KUKA KRL program: chequeo_paleta.src, chequeo_paleta.dat

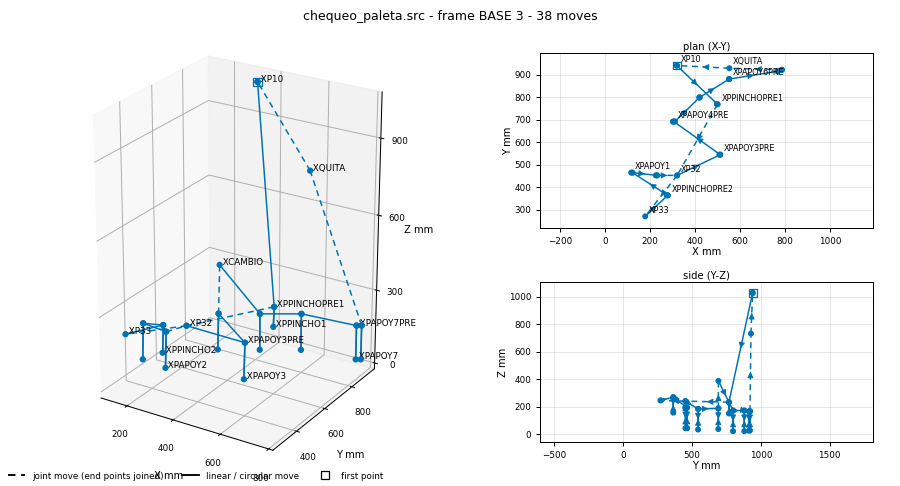
[picture p0: tool path of chequeo_paleta.src in frame BASE 3, 38 of 42 moves have a stored position in this frame; points joined in program order, loops and branches not executed]
--- chequeo_paleta.src ---
&ACCESS RVP
&REL 223
&COMMENT COGER ST121 RACK AZUL
&PARAM EDITMASK = *
&PARAM TEMPLATE = C:\KRC\Roboter\Template\vorgabe
&PARAM DISKPATH = KRC:\R1\Program\MAFELEC
DEF chequeo_paleta( )
;FOLD INI;%{PE}
  ;FOLD BASISTECH INI
    GLOBAL INTERRUPT DECL 3 WHEN $STOPMESS==TRUE DO IR_STOPM ( )
    INTERRUPT ON 3
    BAS (#INITMOV,0 )
  ;ENDFOLD (BASISTECH INI)
;FOLD SPOTTECH INI
USERSPOT(#INIT)
;ENDFOLD (SPOTTECH INI)
;FOLD GRIPPERTECH INI
USER_GRP(0,DUMMY,DUMMY,GDEFAULT)
;ENDFOLD (GRIPPERTECH INI)
;FOLD USER INI
INTERRUPT DECL 26 WHEN I_121R1S102 OR I_121R1S202 DO PARO_RAPIDO ()
INTERRUPT DECL 27 WHEN I_121R1S302 OR I_121R1S402 DO PARO_RAPIDO ()

    ;Make your modifications here

  ;ENDFOLD (USER INI)
;ENDFOLD (INI)
;################################################
; PROYECTO: PLANTA DE BATERIAS
; ROBOT: 121_R1 TERMINATOR
; PROGRAMA: Chequeo_paletas EN ST121
; PALETA MASTER NUMERO 20
; CREADO POR: Borja Carrion
; FECHA: 13-JULIO-2024
;################################################

Empujador(1,"R",FALSE)
Empujador(2,"R",FALSE)

;FOLD PTP HOME Vel=100 % DEFAULT;%{PE}%R 8.3.48,%MKUKATPBASIS,%CMOVE,%VPTP,%P 1:PTP, 2:HOME, 3:, 5:100, 7:DEFAULT
$BWDSTART=FALSE
PDAT_ACT=PDEFAULT
FDAT_ACT=FHOME
BAS(#PTP_PARAMS,100)
$H_POS=XHOME
PTP XHOME
;ENDFOLD
; FOLD ESPERA CONFIRMACION ENTRADA INSPECCION
WAIT FOR I_ST121_INSPECCION
; ENDFOLD

;FOLD PTP POS_ESPERA_ST121 Vel=100 % H Tool[9]:T_Gripper1_Vacio Base[0];%{PE}%R 8.3.48,%MKUKATPBASIS,%CMOVE,%VPTP,%P 1:PTP, 2:POS_ESPERA_ST121, 3:, 5:100, 7:H
$BWDSTART=FALSE
PDAT_ACT=PH
FDAT_ACT=FPOS_ESPERA_ST121
BAS(#PTP_PARAMS,100)
PTP XPOS_ESPERA_ST121
;ENDFOLD

; FOLD ESPERA CONFIRMACION ENTRADA INSPECCION
WAIT FOR I_ST121_INSPECCION
; ENDFOLD

; FOLD CONTROL DE ELEMENTOS MECANICOS EN REPOSO
;CONTROL DE AUSENCIA DE PIEZA EN GRIPPER
IF I_121R1S1000 THEN
HALT
ENDIF

;CONTROL APERTURA GRIPPER

IF (I_121R1S131B==FALSE) OR (I_121R1S132B==FALSE) OR (I_121R1S133B==FALSE) OR (I_121R1S134B==FALSE) THEN
Pines("R")
ENDIF

Empujador(1,"R",TRUE)
Empujador(2,"R",TRUE)
; ENDFOLD

;FOLD PTP P10 CONT Vel=100 % M Tool[9]:T_Gripper1_Vacio Base[3]:ST121;%{PE}%R 8.3.48,%MKUKATPBASIS,%CMOVE,%VPTP,%P 1:PTP, 2:P10, 3:C_DIS, 5:100, 7:M
$BWDSTART=FALSE
PDAT_ACT=PM
FDAT_ACT=FP10
BAS(#PTP_PARAMS,100)
PTP XP10 C_DIS
;ENDFOLD


; ANTES DE EMPEZAR EL CHEQUEO COLOCAR EL UTIL EN LA CLAMPA 3 (QUITAR TONILLO AZUL)
; ABRIR PUERTA DESCARGA MANUAL

; POSICIONES CHEQUEO PINCHOS

; PINCHO 1
;FOLD LIN PPINCHOPRE1 CONT Vel=0.09 m/s M Tool[9]:T_Gripper1_Vacio Base[3]:ST121;%{PE}%R 8.3.48,%MKUKATPBASIS,%CMOVE,%VLIN,%P 1:LIN, 2:PPINCHOPRE1, 3:C_DIS C_DIS, 5:0.09, 7:M
$BWDSTART=FALSE
LDAT_ACT=LM
FDAT_ACT=FPPINCHOPRE1
BAS(#CP_PARAMS,0.09)
LIN XPPINCHOPRE1 C_DIS C_DIS
;ENDFOLD
;FOLD LIN PPINCHO1 CONT Vel=0.02 m/s M Tool[9]:T_Gripper1_Vacio Base[3]:ST121;%{PE}%R 8.3.48,%MKUKATPBASIS,%CMOVE,%VLIN,%P 1:LIN, 2:PPINCHO1, 3:C_DIS C_DIS, 5:0.02, 7:M
$BWDSTART=FALSE
LDAT_ACT=LM
FDAT_ACT=FPPINCHO1
BAS(#CP_PARAMS,0.02)
LIN XPPINCHO1 C_DIS C_DIS
;ENDFOLD
;FOLD WAIT Time=0.5 sec;%{PE}%R 8.3.48,%MKUKATPBASIS,%CWAIT,%VWAIT,%P 3:0.5
WAIT SEC 0.5
;ENDFOLD
;FOLD LIN PPINCHOPRE1 CONT Vel=0.09 m/s M Tool[9]:T_Gripper1_Vacio Base[3]:ST121;%{PE}%R 8.3.48,%MKUKATPBASIS,%CMOVE,%VLIN,%P 1:LIN, 2:PPINCHOPRE1, 3:C_DIS C_DIS, 5:0.09, 7:M
$BWDSTART=FALSE
LDAT_ACT=LM
FDAT_ACT=FPPINCHOPRE1
BAS(#CP_PARAMS,0.09)
LIN XPPINCHOPRE1 C_DIS C_DIS
;ENDFOLD

; PINCHO 2
;FOLD PTP P32 CONT Vel=50 % M Tool[9]:T_Gripper1_Vacio Base[3]:ST121;%{PE}%R 8.3.48,%MKUKATPBASIS,%CMOVE,%VPTP,%P 1:PTP, 2:P32, 3:C_DIS, 5:50, 7:M
$BWDSTART=FALSE
PDAT_ACT=PM
FDAT_ACT=FP32
BAS(#PTP_PARAMS,50)
PTP XP32 C_DIS
;ENDFOLD
;FOLD PTP P33 CONT Vel=50 % M Tool[9]:T_Gripper1_Vacio Base[3]:ST121;%{PE}%R 8.3.48,%MKUKATPBASIS,%CMOVE,%VPTP,%P 1:PTP, 2:P33, 3:C_DIS, 5:50, 7:M
$BWDSTART=FALSE
PDAT_ACT=PM
FDAT_ACT=FP33
BAS(#PTP_PARAMS,50)
PTP XP33 C_DIS
;ENDFOLD
;FOLD LIN PPINCHOPRE2 CONT Vel=0.09 m/s M Tool[9]:T_Gripper1_Vacio Base[3]:ST121;%{PE}%R 8.3.48,%MKUKATPBASIS,%CMOVE,%VLIN,%P 1:LIN, 2:PPINCHOPRE2, 3:C_DIS C_DIS, 5:0.09, 7:M
$BWDSTART=FALSE
LDAT_ACT=LM
FDAT_ACT=FPPINCHOPRE2
BAS(#CP_PARAMS,0.09)
LIN XPPINCHOPRE2 C_DIS C_DIS
;ENDFOLD
;FOLD LIN PPINCHO2 CONT Vel=0.02 m/s M Tool[9]:T_Gripper1_Vacio Base[3]:ST121;%{PE}%R 8.3.48,%MKUKATPBASIS,%CMOVE,%VLIN,%P 1:LIN, 2:PPINCHO2, 3:C_DIS C_DIS, 5:0.02, 7:M
$BWDSTART=FALSE
LDAT_ACT=LM
FDAT_ACT=FPPINCHO2
BAS(#CP_PARAMS,0.02)
LIN XPPINCHO2 C_DIS C_DIS
;ENDFOLD
;FOLD WAIT Time=0.5 sec;%{PE}%R 8.3.48,%MKUKATPBASIS,%CWAIT,%VWAIT,%P 3:0.5
WAIT SEC 0.5
;ENDFOLD
;FOLD LIN PPINCHOPRE2 CONT Vel=0.09 m/s M Tool[9]:T_Gripper1_Vacio Base[3]:ST121;%{PE}%R 8.3.48,%MKUKATPBASIS,%CMOVE,%VLIN,%P 1:LIN, 2:PPINCHOPRE2, 3:C_DIS C_DIS, 5:0.09, 7:M
$BWDSTART=FALSE
LDAT_ACT=LM
FDAT_ACT=FPPINCHOPRE2
BAS(#CP_PARAMS,0.09)
LIN XPPINCHOPRE2 C_DIS C_DIS
;ENDFOLD

;FOLD WAIT Time=1 sec;%{PE}%R 8.3.48,%MKUKATPBASIS,%CWAIT,%VWAIT,%P 3:1
WAIT SEC 1
;ENDFOLD


; POSICIONES CHEQUEO APOYOS
; APOYO 1
;FOLD LIN PAPOY1PRE CONT Vel=0.09 m/s M Tool[9]:T_Gripper1_Vacio Base[3]:ST121;%{PE}%R 8.3.48,%MKUKATPBASIS,%CMOVE,%VLIN,%P 1:LIN, 2:PAPOY1PRE, 3:C_DIS C_DIS, 5:0.09, 7:M
$BWDSTART=FALSE
LDAT_ACT=LM
FDAT_ACT=FPAPOY1PRE
BAS(#CP_PARAMS,0.09)
LIN XPAPOY1PRE C_DIS C_DIS
;ENDFOLD
;FOLD LIN PAPOY1 Vel=0.02 m/s M Tool[9]:T_Gripper1_Vacio Base[3]:ST121;%{PE}%R 8.3.48,%MKUKATPBASIS,%CMOVE,%VLIN,%P 1:LIN, 2:PAPOY1, 3:, 5:0.02, 7:M
$BWDSTART=FALSE
LDAT_ACT=LM
FDAT_ACT=FPAPOY1
BAS(#CP_PARAMS,0.02)
LIN XPAPOY1
;ENDFOLD
;FOLD WAIT Time=0.5 sec;%{PE}%R 8.3.48,%MKUKATPBASIS,%CWAIT,%VWAIT,%P 3:0.5
WAIT SEC 0.5
;ENDFOLD
;FOLD LIN PAPOY1PRE CONT Vel=0.09 m/s M Tool[9]:T_Gripper1_Vacio Base[3]:ST121;%{PE}%R 8.3.48,%MKUKATPBASIS,%CMOVE,%VLIN,%P 1:LIN, 2:PAPOY1PRE, 3:C_DIS C_DIS, 5:0.09, 7:M
$BWDSTART=FALSE
LDAT_ACT=LM
FDAT_ACT=FPAPOY1PRE
BAS(#CP_PARAMS,0.09)
LIN XPAPOY1PRE C_DIS C_DIS
;ENDFOLD

; APOYO 2
;FOLD LIN PAPOY2PRE CONT Vel=0.09 m/s M Tool[9]:T_Gripper1_Vacio Base[3]:ST121;%{PE}%R 8.3.48,%MKUKATPBASIS,%CMOVE,%VLIN,%P 1:LIN, 2:PAPOY2PRE, 3:C_DIS C_DIS, 5:0.09, 7:M
$BWDSTART=FALSE
LDAT_ACT=LM
FDAT_ACT=FPAPOY2PRE
BAS(#CP_PARAMS,0.09)
LIN XPAPOY2PRE C_DIS C_DIS
;ENDFOLD
;FOLD LIN PAPOY2 CONT Vel=0.02 m/s M Tool[9]:T_Gripper1_Vacio Base[3]:ST121;%{PE}%R 8.3.48,%MKUKATPBASIS,%CMOVE,%VLIN,%P 1:LIN, 2:PAPOY2, 3:C_DIS C_DIS, 5:0.02, 7:M
$BWDSTART=FALSE
LDAT_ACT=LM
FDAT_ACT=FPAPOY2
BAS(#CP_PARAMS,0.02)
LIN XPAPOY2 C_DIS C_DIS
;ENDFOLD
;FOLD WAIT Time=0.5 sec;%{PE}%R 8.3.48,%MKUKATPBASIS,%CWAIT,%VWAIT,%P 3:0.5
WAIT SEC 0.5
;ENDFOLD
;FOLD LIN PAPOY2PRE CONT Vel=0.09 m/s M Tool[9]:T_Gripper1_Vacio Base[3]:ST121;%{PE}%R 8.3.48,%MKUKATPBASIS,%CMOVE,%VLIN,%P 1:LIN, 2:PAPOY2PRE, 3:C_DIS C_DIS, 5:0.09, 7:M
$BWDSTART=FALSE
LDAT_ACT=LM
FDAT_ACT=FPAPOY2PRE
BAS(#CP_PARAMS,0.09)
LIN XPAPOY2PRE C_DIS C_DIS
;ENDFOLD

;FOLD PTP P39 CONT Vel=50 % M Tool[9]:T_Gripper1_Vacio Base[3]:ST121;%{PE}%R 8.3.48,%MKUKATPBASIS,%CMOVE,%VPTP,%P 1:PTP, 2:P39, 3:C_DIS, 5:50, 7:M
$BWDSTART=FALSE
PDAT_ACT=PM
FDAT_ACT=FP39
BAS(#PTP_PARAMS,50)
PTP XP39 C_DIS
;ENDFOLD


; APOYO 3
;FOLD LIN PAPOY3PRE CONT Vel=0.09 m/s M Tool[9]:T_Gripper1_Vacio Base[3]:ST121;%{PE}%R 8.3.48,%MKUKATPBASIS,%CMOVE,%VLIN,%P 1:LIN, 2:PAPOY3PRE, 3:C_DIS C_DIS, 5:0.09, 7:M
$BWDSTART=FALSE
LDAT_ACT=LM
FDAT_ACT=FPAPOY3PRE
BAS(#CP_PARAMS,0.09)
LIN XPAPOY3PRE C_DIS C_DIS
;ENDFOLD
;FOLD LIN PAPOY3 CONT Vel=0.02 m/s M Tool[9]:T_Gripper1_Vacio Base[3]:ST121;%{PE}%R 8.3.48,%MKUKATPBASIS,%CMOVE,%VLIN,%P 1:LIN, 2:PAPOY3, 3:C_DIS C_DIS, 5:0.02, 7:M
$BWDSTART=FALSE
LDAT_ACT=LM
FDAT_ACT=FPAPOY3
BAS(#CP_PARAMS,0.02)
LIN XPAPOY3 C_DIS C_DIS
;ENDFOLD
;FOLD WAIT Time=0.5 sec;%{PE}%R 8.3.48,%MKUKATPBASIS,%CWAIT,%VWAIT,%P 3:0.5
WAIT SEC 0.5
;ENDFOLD
;FOLD LIN PAPOY3PRE CONT Vel=0.09 m/s M Tool[9]:T_Gripper1_Vacio Base[3]:ST121;%{PE}%R 8.3.48,%MKUKATPBASIS,%CMOVE,%VLIN,%P 1:LIN, 2:PAPOY3PRE, 3:C_DIS C_DIS, 5:0.09, 7:M
$BWDSTART=FALSE
LDAT_ACT=LM
FDAT_ACT=FPAPOY3PRE
BAS(#CP_PARAMS,0.09)
LIN XPAPOY3PRE C_DIS C_DIS
;ENDFOLD

; APOYO 4
;FOLD LIN PAPOY4PRE CONT Vel=0.09 m/s M Tool[9]:T_Gripper1_Vacio Base[3]:ST121;%{PE}%R 8.3.48,%MKUKATPBASIS,%CMOVE,%VLIN,%P 1:LIN, 2:PAPOY4PRE, 3:C_DIS C_DIS, 5:0.09, 7:M
$BWDSTART=FALSE
LDAT_ACT=LM
FDAT_ACT=FPAPOY4PRE
BAS(#CP_PARAMS,0.09)
LIN XPAPOY4PRE C_DIS C_DIS
;ENDFOLD
;FOLD LIN PAPOY4 CONT Vel=0.02 m/s M Tool[9]:T_Gripper1_Vacio Base[3]:ST121;%{PE}%R 8.3.48,%MKUKATPBASIS,%CMOVE,%VLIN,%P 1:LIN, 2:PAPOY4, 3:C_DIS C_DIS, 5:0.02, 7:M
$BWDSTART=FALSE
LDAT_ACT=LM
FDAT_ACT=FPAPOY4
BAS(#CP_PARAMS,0.02)
LIN XPAPOY4 C_DIS C_DIS
;ENDFOLD
;FOLD WAIT Time=0.5 sec;%{PE}%R 8.3.48,%MKUKATPBASIS,%CWAIT,%VWAIT,%P 3:0.5
WAIT SEC 0.5
;ENDFOLD
;FOLD LIN PAPOY4PRE Vel=0.09 m/s M Tool[9]:T_Gripper1_Vacio Base[3]:ST121;%{PE}%R 8.3.48,%MKUKATPBASIS,%CMOVE,%VLIN,%P 1:LIN, 2:PAPOY4PRE, 3:, 5:0.09, 7:M
$BWDSTART=FALSE
LDAT_ACT=LM
FDAT_ACT=FPAPOY4PRE
BAS(#CP_PARAMS,0.09)
LIN XPAPOY4PRE
;ENDFOLD

;QUITA UTIL CLAMPA 3 (TORNILLO AZUL)

;POSICION PARA CAMBIAR UTIL A CLAMPA 1 (TORNILLO AZUL)
;FOLD PTP CAMBIO CONT Vel=50 % H Tool[9]:T_Gripper1_Vacio Base[3]:ST121;%{PE}%R 8.3.48,%MKUKATPBASIS,%CMOVE,%VPTP,%P 1:PTP, 2:CAMBIO, 3:C_DIS, 5:50, 7:H
$BWDSTART=FALSE
PDAT_ACT=PH
FDAT_ACT=FCAMBIO
BAS(#PTP_PARAMS,50)
PTP XCAMBIO C_DIS
;ENDFOLD
;FOLD WAIT Time=5 sec;%{PE}%R 8.3.48,%MKUKATPBASIS,%CWAIT,%VWAIT,%P 3:5
WAIT SEC 5
;ENDFOLD

; APOYO 5
;FOLD LIN PAPOY5PRE CONT Vel=0.09 m/s M Tool[9]:T_Gripper1_Vacio Base[3]:ST121;%{PE}%R 8.3.48,%MKUKATPBASIS,%CMOVE,%VLIN,%P 1:LIN, 2:PAPOY5PRE, 3:C_DIS C_DIS, 5:0.09, 7:M
$BWDSTART=FALSE
LDAT_ACT=LM
FDAT_ACT=FPAPOY5PRE
BAS(#CP_PARAMS,0.09)
LIN XPAPOY5PRE C_DIS C_DIS
;ENDFOLD
;FOLD LIN PAPOY5 CONT Vel=0.02 m/s M Tool[9]:T_Gripper1_Vacio Base[3]:ST121;%{PE}%R 8.3.48,%MKUKATPBASIS,%CMOVE,%VLIN,%P 1:LIN, 2:PAPOY5, 3:C_DIS C_DIS, 5:0.02, 7:M
$BWDSTART=FALSE
LDAT_ACT=LM
FDAT_ACT=FPAPOY5
BAS(#CP_PARAMS,0.02)
LIN XPAPOY5 C_DIS C_DIS
;ENDFOLD
;FOLD WAIT Time=0.5 sec;%{PE}%R 8.3.48,%MKUKATPBASIS,%CWAIT,%VWAIT,%P 3:0.5
WAIT SEC 0.5
;ENDFOLD
;FOLD LIN PAPOY5PRE CONT Vel=0.09 m/s M Tool[9]:T_Gripper1_Vacio Base[3]:ST121;%{PE}%R 8.3.48,%MKUKATPBASIS,%CMOVE,%VLIN,%P 1:LIN, 2:PAPOY5PRE, 3:C_DIS C_DIS, 5:0.09, 7:M
$BWDSTART=FALSE
LDAT_ACT=LM
FDAT_ACT=FPAPOY5PRE
BAS(#CP_PARAMS,0.09)
LIN XPAPOY5PRE C_DIS C_DIS
;ENDFOLD

; APOYO 6
;FOLD LIN PAPOY6PRE CONT Vel=0.09 m/s M Tool[9]:T_Gripper1_Vacio Base[3]:ST121;%{PE}%R 8.3.48,%MKUKATPBASIS,%CMOVE,%VLIN,%P 1:LIN, 2:PAPOY6PRE, 3:C_DIS C_DIS, 5:0.09, 7:M
$BWDSTART=FALSE
LDAT_ACT=LM
FDAT_ACT=FPAPOY6PRE
BAS(#CP_PARAMS,0.09)
LIN XPAPOY6PRE C_DIS C_DIS
;ENDFOLD
;FOLD LIN PAPOY6 CONT Vel=0.02 m/s M Tool[9]:T_Gripper1_Vacio Base[3]:ST121;%{PE}%R 8.3.48,%MKUKATPBASIS,%CMOVE,%VLIN,%P 1:LIN, 2:PAPOY6, 3:C_DIS C_DIS, 5:0.02, 7:M
$BWDSTART=FALSE
LDAT_ACT=LM
FDAT_ACT=FPAPOY6
BAS(#CP_PARAMS,0.02)
LIN XPAPOY6 C_DIS C_DIS
;ENDFOLD
;FOLD WAIT Time=0.5 sec;%{PE}%R 8.3.48,%MKUKATPBASIS,%CWAIT,%VWAIT,%P 3:0.5
WAIT SEC 0.5
;ENDFOLD
;FOLD LIN PAPOY6PRE Vel=0.09 m/s M Tool[9]:T_Gripper1_Vacio Base[3]:ST121;%{PE}%R 8.3.48,%MKUKATPBASIS,%CMOVE,%VLIN,%P 1:LIN, 2:PAPOY6PRE, 3:, 5:0.09, 7:M
$BWDSTART=FALSE
LDAT_ACT=LM
FDAT_ACT=FPAPOY6PRE
BAS(#CP_PARAMS,0.09)
LIN XPAPOY6PRE
;ENDFOLD


; APOYO 7
;FOLD LIN PAPOY7PRE CONT Vel=0.09 m/s M Tool[9]:T_Gripper1_Vacio Base[3]:ST121;%{PE}%R 8.3.48,%MKUKATPBASIS,%CMOVE,%VLIN,%P 1:LIN, 2:PAPOY7PRE, 3:C_DIS C_DIS, 5:0.09, 7:M
$BWDSTART=FALSE
LDAT_ACT=LM
FDAT_ACT=FPAPOY7PRE
BAS(#CP_PARAMS,0.09)
LIN XPAPOY7PRE C_DIS C_DIS
;ENDFOLD
;FOLD LIN PAPOY7 CONT Vel=0.02 m/s M Tool[9]:T_Gripper1_Vacio Base[3]:ST121;%{PE}%R 8.3.48,%MKUKATPBASIS,%CMOVE,%VLIN,%P 1:LIN, 2:PAPOY7, 3:C_DIS C_DIS, 5:0.02, 7:M
$BWDSTART=FALSE
LDAT_ACT=LM
FDAT_ACT=FPAPOY7
BAS(#CP_PARAMS,0.02)
LIN XPAPOY7 C_DIS C_DIS
;ENDFOLD
;FOLD WAIT Time=0.5 sec;%{PE}%R 8.3.48,%MKUKATPBASIS,%CWAIT,%VWAIT,%P 3:0.5
WAIT SEC 0.5
;ENDFOLD
;FOLD LIN PAPOY7PRE CONT Vel=0.09 m/s M Tool[9]:T_Gripper1_Vacio Base[3]:ST121;%{PE}%R 8.3.48,%MKUKATPBASIS,%CMOVE,%VLIN,%P 1:LIN, 2:PAPOY7PRE, 3:C_DIS C_DIS, 5:0.09, 7:M
$BWDSTART=FALSE
LDAT_ACT=LM
FDAT_ACT=FPAPOY7PRE
BAS(#CP_PARAMS,0.09)
LIN XPAPOY7PRE C_DIS C_DIS
;ENDFOLD

; APOYO 8
;FOLD LIN PAPOY8PRE CONT Vel=0.09 m/s M Tool[9]:T_Gripper1_Vacio Base[3]:ST121;%{PE}%R 8.3.48,%MKUKATPBASIS,%CMOVE,%VLIN,%P 1:LIN, 2:PAPOY8PRE, 3:C_DIS C_DIS, 5:0.09, 7:M
$BWDSTART=FALSE
LDAT_ACT=LM
FDAT_ACT=FPAPOY8PRE
BAS(#CP_PARAMS,0.09)
LIN XPAPOY8PRE C_DIS C_DIS
;ENDFOLD
;FOLD LIN PAPOY8 CONT Vel=0.02 m/s M Tool[9]:T_Gripper1_Vacio Base[3]:ST121;%{PE}%R 8.3.48,%MKUKATPBASIS,%CMOVE,%VLIN,%P 1:LIN, 2:PAPOY8, 3:C_DIS C_DIS, 5:0.02, 7:M
$BWDSTART=FALSE
LDAT_ACT=LM
FDAT_ACT=FPAPOY8
BAS(#CP_PARAMS,0.02)
LIN XPAPOY8 C_DIS C_DIS
;ENDFOLD
;FOLD WAIT Time=0.5 sec;%{PE}%R 8.3.48,%MKUKATPBASIS,%CWAIT,%VWAIT,%P 3:0.5
WAIT SEC 0.5
;ENDFOLD
;FOLD LIN PAPOY8PRE Vel=0.09 m/s M Tool[9]:T_Gripper1_Vacio Base[3]:ST121;%{PE}%R 8.3.48,%MKUKATPBASIS,%CMOVE,%VLIN,%P 1:LIN, 2:PAPOY8PRE, 3:, 5:0.09, 7:M
$BWDSTART=FALSE
LDAT_ACT=LM
FDAT_ACT=FPAPOY8PRE
BAS(#CP_PARAMS,0.09)
LIN XPAPOY8PRE
;ENDFOLD

;POSICION PARA QUTAR UTIL CLAMPA 1 (TORNILLO AZUL)
;FOLD PTP QUITA CONT Vel=50 % H Tool[9]:T_Gripper1_Vacio Base[3]:ST121;%{PE}%R 8.3.48,%MKUKATPBASIS,%CMOVE,%VPTP,%P 1:PTP, 2:QUITA, 3:C_DIS, 5:50, 7:H
$BWDSTART=FALSE
PDAT_ACT=PH
FDAT_ACT=FQUITA
BAS(#PTP_PARAMS,50)
PTP XQUITA C_DIS
;ENDFOLD

;FOLD WAIT Time=5 sec;%{PE}%R 8.3.48,%MKUKATPBASIS,%CWAIT,%VWAIT,%P 3:5
WAIT SEC 5
;ENDFOLD
;FOLD PTP P38 CONT Vel=100 % M Tool[9]:T_Gripper1_Vacio Base[3]:ST121;%{PE}%R 8.3.48,%MKUKATPBASIS,%CMOVE,%VPTP,%P 1:PTP, 2:P38, 3:C_DIS, 5:100, 7:M
$BWDSTART=FALSE
PDAT_ACT=PM
FDAT_ACT=FP38
BAS(#PTP_PARAMS,100)
PTP XP38 C_DIS
;ENDFOLD

;FOLD PTP POS_SOBRE_ST121 Vel=50 % H Tool[9]:T_Gripper1_Vacio Base[3]:ST121;%{PE}%R 8.3.48,%MKUKATPBASIS,%CMOVE,%VPTP,%P 1:PTP, 2:POS_SOBRE_ST121, 3:, 5:50, 7:H
$BWDSTART=FALSE
PDAT_ACT=PH
FDAT_ACT=FPOS_SOBRE_ST121
BAS(#PTP_PARAMS,50)
PTP XPOS_SOBRE_ST121
;ENDFOLD


;POSICION AREA 3 LIBRE
;FOLD PTP POS_ESPERA_ST122 Vel=100 % H Tool[9]:T_Gripper1_Vacio Base[0];%{PE}%R 8.3.48,%MKUKATPBASIS,%CMOVE,%VPTP,%P 1:PTP, 2:POS_ESPERA_ST122, 3:, 5:100, 7:H
$BWDSTART=FALSE
PDAT_ACT=PH
FDAT_ACT=FPOS_ESPERA_ST122
BAS(#PTP_PARAMS,100)
PTP XPOS_ESPERA_ST122
;ENDFOLD

;LIBERA AREA 3, TRANSPORTE BATERIAS
O_AREL_3=TRUE


;FOLD PTP HOME Vel=100 % DEFAULT;%{PE}%R 8.3.48,%MKUKATPBASIS,%CMOVE,%VPTP,%P 1:PTP, 2:HOME, 3:, 5:100, 7:DEFAULT
$BWDSTART=FALSE
PDAT_ACT=PDEFAULT
FDAT_ACT=FHOME
BAS(#PTP_PARAMS,100)
$H_POS=XHOME
PTP XHOME
;ENDFOLD

END
DEF PARO_RAPIDO ()
BRAKE F
END

--- chequeo_paleta.dat ---
&ACCESS RVP
&REL 223
&COMMENT COGER ST121 RACK AZUL
&PARAM EDITMASK = *
&PARAM TEMPLATE = C:\KRC\Roboter\Template\vorgabe
&PARAM DISKPATH = KRC:\R1\Program\MAFELEC
DEFDAT  chequeo_paleta
;FOLD EXTERNAL DECLARATIONS;%{PE}%MKUKATPBASIS,%CEXT,%VCOMMON,%P
;FOLD GRIPPERTECH EXT
EXT  H50 (INT  :IN,INT  :IN,INT  :IN,GRP_TYP  :IN )
;ENDFOLD (GRIPPERTECH EXT)
;FOLD SPOTTECH EXT
EXT  USERSPOT (S_COMMAND  :IN,SPOT_TYPE  :IN )
;ENDFOLD (SPOTTECH EXT)
;FOLD BASISTECH EXT;%{PE}%MKUKATPBASIS,%CEXT,%VEXT,%P
EXT  BAS (BAS_COMMAND  :IN,REAL  :IN )
DECL INT SUCCESS
;ENDFOLD (BASISTECH EXT)
;FOLD USER EXT;%{E}%MKUKATPUSER,%CEXT,%VEXT,%P
;Make your modifications here

;ENDFOLD (USER EXT)
;ENDFOLD (EXTERNAL DECLARATIONS)
DECL BASIS_SUGG_T LAST_BASIS={POINT1[] "QUITA                   ",POINT2[] "QUITA                   ",CP_PARAMS[] "M                       ",PTP_PARAMS[] "H                       ",CONT[] "C_DIS                   ",CP_VEL[] "0.09                    ",PTP_VEL[] "50                      ",SYNC_PARAMS[] "SYNCDAT                 ",SPL_NAME[] "S0                      ",A_PARAMS[] "ADAT0                   "}
DECL PDAT PH={VEL 100.000,ACC 100.000,APO_DIST 100.000,APO_MODE #CDIS,GEAR_JERK 50.0000,EXAX_IGN 0}
DECL E6POS XP10={X 318.805969,Y 940.468872,Z 1027.99695,A -176.544083,B 30.8923950,C -165.320572,S 2,T 2,E1 0.0,E2 0.0,E3 0.0,E4 0.0,E5 0.0,E6 0.0}
DECL FDAT FP10={TOOL_NO 9,BASE_NO 3,IPO_FRAME #BASE,POINT2[] " ",TQ_STATE FALSE}
DECL E6POS XP20={X 312.450226,Y 675.070,Z 73.4258270,A -0.219463497,B -0.287549138,C -179.748962,S 2,T 42,E1 0.0,E2 0.0,E3 0.0,E4 0.0,E5 0.0,E6 0.0}
DECL FDAT FP20={TOOL_NO 9,BASE_NO 3,IPO_FRAME #BASE,POINT2[] " ",TQ_STATE FALSE}
DECL E6POS XPOS_COGER_ST121={X 364.233917,Y 680.820,Z 35.4071388,A -0.219463244,B -0.287549198,C -179.748962,S 2,T 42,E1 0.0,E2 0.0,E3 0.0,E4 0.0,E5 0.0,E6 0.0}
DECL FDAT FPos_Coger_ST121={TOOL_NO 9,BASE_NO 3,IPO_FRAME #BASE,POINT2[] " ",TQ_STATE FALSE}
DECL PDAT PM={VEL 100.000,ACC 50.0000,APO_DIST 50.0000,APO_MODE #CDIS,GEAR_JERK 50.0000,EXAX_IGN 0}
DECL E6POS XPOS_ESPERA_ST121={X 1597.05444,Y -395.116150,Z 1941.31274,A -176.307449,B 30.3077869,C -171.065643,S 2,T 10,E1 0.0,E2 0.0,E3 0.0,E4 0.0,E5 0.0,E6 0.0}
DECL FDAT FPOS_ESPERA_ST121={TOOL_NO 9,BASE_NO 0,IPO_FRAME #BASE,POINT2[] " ",TQ_STATE FALSE}
DECL LDAT LM={VEL 2.00000,ACC 25.0000,APO_DIST 100.000,APO_FAC 50.0000,AXIS_VEL 100.000,AXIS_ACC 100.000,ORI_TYP #VAR,CIRC_TYP #BASE,JERK_FAC 50.0000,GEAR_JERK 50.0000,EXAX_IGN 0}
DECL E6POS XPOS_SOBRE_ST121={X 318.805969,Y 940.468872,Z 1027.99695,A -176.544083,B 30.8923950,C -165.320572,S 2,T 2,E1 0.0,E2 0.0,E3 0.0,E4 0.0,E5 0.0,E6 0.0}
DECL FDAT FPOS_SOBRE_ST121={TOOL_NO 9,BASE_NO 3,IPO_FRAME #BASE,POINT2[] " ",TQ_STATE FALSE}
DECL E6POS XPOS_SOBRE_ST122={X 1790.32410,Y 1.34322268E-13,Z 1909.62585,A -180.000,B 89.9853210,C -180.000,S 2,T 3,E1 0.0,E2 0.0,E3 0.0,E4 0.0,E5 0.0,E6 0.0}
DECL FDAT FPOS_SOBRE_ST122={TOOL_NO 9,BASE_NO 3,IPO_FRAME #BASE,POINT2[] " ",TQ_STATE FALSE}
DECL E6POS XP30={X 158.918106,Y 1091.44617,Z 654.405884,A 42.3399849,B -0.235063374,C -179.753174,S 2,T 42,E1 0.0,E2 0.0,E3 0.0,E4 0.0,E5 0.0,E6 0.0}
DECL FDAT FP30={TOOL_NO 11,BASE_NO 3,IPO_FRAME #BASE,POINT2[] " ",TQ_STATE FALSE}
DECL E6POS XP40={X -0.0319372341,Y -2.62910700,Z -362.053223,A -0.00123304490,B -0.0257057231,C 0.00384289422,S 2,T 10,E1 0.0,E2 0.0,E3 0.0,E4 0.0,E5 0.0,E6 0.0}
DECL FDAT FP40={TOOL_NO 11,BASE_NO 3,IPO_FRAME #BASE,POINT2[] " ",TQ_STATE FALSE}
DECL E6POS XPOS_AREA_3_LIBRE={X 1597.05457,Y -395.116180,Z 1941.31274,A -176.307449,B 30.3077888,C -171.065643,S 2,T 10,E1 0.0,E2 0.0,E3 0.0,E4 0.0,E5 0.0,E6 0.0}
DECL FDAT FPOS_AREA_3_LIBRE={TOOL_NO 9,BASE_NO 3,IPO_FRAME #BASE,POINT2[] " ",TQ_STATE FALSE}
DECL GRP_SUGG_T LAST_GRP={NUMBER[] "1                       ",STATE[] "1                       ",PARAMS[] "GDAT0                   "}
DECL LDAT LL={VEL 2.00000,ACC 25.0000,APO_DIST 100.000,APO_FAC 50.0000,AXIS_VEL 100.000,AXIS_ACC 100.000,ORI_TYP #VAR,CIRC_TYP #BASE,JERK_FAC 50.0000,GEAR_JERK 50.0000,EXAX_IGN 0}
DECL PDAT PL={VEL 100.000,ACC 25.0000,APO_DIST 50.0000,APO_MODE #CDIS,GEAR_JERK 50.0000,EXAX_IGN 0}
DECL E6POS XP0={X 364.480164,Y 681.182129,Z 388.540192,A -0.219463348,B -0.287549168,C -179.748962,S 2,T 42,E1 0.0,E2 0.0,E3 0.0,E4 0.0,E5 0.0,E6 0.0}
DECL FDAT FP0={TOOL_NO 9,BASE_NO 3,IPO_FRAME #BASE,POINT2[] " ",TQ_STATE FALSE}
DECL E6POS XP1={X 364.233917,Y 677.270142,Z 82.2082901,A -0.219467312,B -0.287552059,C -179.748962,S 2,T 42,E1 0.0,E2 0.0,E3 0.0,E4 0.0,E5 0.0,E6 0.0}
DECL FDAT FP1={TOOL_NO 9,BASE_NO 3,IPO_FRAME #BASE,POINT2[] " ",TQ_STATE FALSE}
DECL E6POS XPos_Coger_Verde_ST121={X 364.233917,Y 680.820,Z 35.4071388,A -0.219467372,B -0.287552029,C -179.748962,S 2,T 42,E1 0.0,E2 0.0,E3 0.0,E4 0.0,E5 0.0,E6 0.0}
DECL FDAT FPos_Coger_Verde_ST121={TOOL_NO 9,BASE_NO 3,IPO_FRAME #BASE,POINT2[] " ",TQ_STATE FALSE}
DECL E6POS XCOGER_ST121_INSP={X 312.450226,Y 675.070,Z 31.2908478,A -0.219463453,B -0.287549138,C -179.748962,S 2,T 42,E1 0.0,E2 0.0,E3 0.0,E4 0.0,E5 0.0,E6 0.0}
DECL FDAT FCoger_ST121_INSP={TOOL_NO 9,BASE_NO 3,IPO_FRAME #BASE,POINT2[] " ",TQ_STATE FALSE}
DECL E6POS XPOS_ESPERA_ST122={X 1597.05444,Y -395.116150,Z 1941.31274,A -176.307449,B 30.3077869,C -171.065643,S 2,T 10,E1 0.0,E2 0.0,E3 0.0,E4 0.0,E5 0.0,E6 0.0}
DECL FDAT FPOS_ESPERA_ST122={TOOL_NO 9,BASE_NO 0,IPO_FRAME #BASE,POINT2[] " ",TQ_STATE FALSE}
DECL E6POS XP31={X 496.711304,Y 768.397461,Z 151.694839,A -177.583694,B -2.05908513,C 179.837936,S 2,T 2,E1 0.0,E2 0.0,E3 0.0,E4 0.0,E5 0.0,E6 0.0}
DECL FDAT FP31={TOOL_NO 9,BASE_NO 3,IPO_FRAME #BASE,POINT2[] " ",TQ_STATE FALSE}
DECL E6POS XP32={X 320.366150,Y 452.067413,Z 241.559097,A 154.607697,B -1.89703083,C -179.182938,S 2,T 34,E1 0.0,E2 0.0,E3 0.0,E4 0.0,E5 0.0,E6 0.0}
DECL FDAT FP32={TOOL_NO 9,BASE_NO 3,IPO_FRAME #BASE,POINT2[] " ",TQ_STATE FALSE}
DECL E6POS XP33={X 178.176437,Y 270.095551,Z 246.496567,A 110.042107,B -0.778272212,C -178.086685,S 2,T 34,E1 0.0,E2 0.0,E3 0.0,E4 0.0,E5 0.0,E6 0.0}
DECL FDAT FP33={TOOL_NO 9,BASE_NO 3,IPO_FRAME #BASE,POINT2[] " ",TQ_STATE FALSE}
DECL E6POS XP34={X -150.954285,Y 165.473572,Z 618.738037,A -179.160065,B 43.8682137,C -176.870,S 2,T 10,E1 0.0,E2 0.0,E3 0.0,E4 0.0,E5 0.0,E6 0.0}
DECL FDAT FP34={TOOL_NO 9,BASE_NO 3,IPO_FRAME #BASE,POINT2[] " ",TQ_STATE FALSE}
DECL E6POS XP35={X -140.190475,Y 628.990662,Z 600.472900,A -179.160065,B 43.8682137,C -176.870,S 2,T 10,E1 0.0,E2 0.0,E3 0.0,E4 0.0,E5 0.0,E6 0.0}
DECL FDAT FP35={TOOL_NO 9,BASE_NO 3,IPO_FRAME #BASE,POINT2[] " ",TQ_STATE FALSE}
DECL E6POS XP36={X -130.254105,Y 1132.55237,Z 623.664185,A -179.158569,B 43.8791924,C -176.869125,S 2,T 34,E1 0.0,E2 0.0,E3 0.0,E4 0.0,E5 0.0,E6 0.0}
DECL FDAT FP36={TOOL_NO 9,BASE_NO 3,IPO_FRAME #BASE,POINT2[] " ",TQ_STATE FALSE}
DECL E6POS XP33_ENLACE={X -225.899948,Y 1138.68835,Z 723.022644,A -179.158569,B 43.8791847,C -176.869125,S 2,T 34,E1 0.0,E2 0.0,E3 0.0,E4 0.0,E5 0.0,E6 0.0}
DECL FDAT FP33_ENLACE={TOOL_NO 9,BASE_NO 3,IPO_FRAME #BASE,POINT2[] " ",TQ_STATE FALSE}
DECL E6POS XPPINCHO1={X 496.711304,Y 768.397461,Z 151.694839,A -177.583694,B -2.05908513,C 179.837936,S 2,T 2,E1 0.0,E2 0.0,E3 0.0,E4 0.0,E5 0.0,E6 0.0}
DECL FDAT FPPINCHO1={TOOL_NO 9,BASE_NO 3,IPO_FRAME #BASE,POINT2[] " ",TQ_STATE FALSE}
DECL E6POS XPPINCHOPRE={X 499.695221,Y 768.288818,Z 234.487564,A -177.583694,B -2.05908513,C 179.837936,S 2,T 2,E1 0.0,E2 0.0,E3 0.0,E4 0.0,E5 0.0,E6 0.0}
DECL FDAT FPPINCHOPRE={TOOL_NO 9,BASE_NO 3,IPO_FRAME #BASE,POINT2[] " ",TQ_STATE FALSE}
DECL E6POS XPPINCHOPRE1={X 499.695221,Y 768.288818,Z 234.487564,A -177.583694,B -2.05908513,C 179.837936,S 2,T 2,E1 0.0,E2 0.0,E3 0.0,E4 0.0,E5 0.0,E6 0.0}
DECL FDAT FPPINCHOPRE1={TOOL_NO 9,BASE_NO 3,IPO_FRAME #BASE,POINT2[] " ",TQ_STATE FALSE}
DECL E6POS XPPINCHOPRE2={X 278.351349,Y 363.439819,Z 270.109253,A 90.9893951,B -0.110822536,C -177.937485,S 2,T 34,E1 0.0,E2 0.0,E3 0.0,E4 0.0,E5 0.0,E6 0.0}
DECL FDAT FPPINCHOPRE2={TOOL_NO 9,BASE_NO 3,IPO_FRAME #BASE,POINT2[] " ",TQ_STATE FALSE}
DECL E6POS XPPINCHO2={X 274.299774,Y 363.587311,Z 157.694733,A 90.9893951,B -0.110822521,C -177.937485,S 2,T 34,E1 0.0,E2 0.0,E3 0.0,E4 0.0,E5 0.0,E6 0.0}
DECL FDAT FPPINCHO2={TOOL_NO 9,BASE_NO 3,IPO_FRAME #BASE,POINT2[] " ",TQ_STATE FALSE}
DECL E6POS XPPINCHOPRE3={X 212.242874,Y 214.835464,Z 245.075195,A 105.754181,B -0.633007586,C -178.033859,S 2,T 34,E1 0.0,E2 0.0,E3 0.0,E4 0.0,E5 0.0,E6 0.0}
DECL FDAT FPPINCHOPRE3={TOOL_NO 9,BASE_NO 3,IPO_FRAME #BASE,POINT2[] " ",TQ_STATE FALSE}
DECL E6POS XP37={X 320.366150,Y 452.067413,Z 241.559097,A 154.607697,B -1.89703083,C -179.182938,S 2,T 34,E1 0.0,E2 0.0,E3 0.0,E4 0.0,E5 0.0,E6 0.0}
DECL FDAT FP37={TOOL_NO 9,BASE_NO 3,IPO_FRAME #BASE,POINT2[] " ",TQ_STATE FALSE}
DECL E6POS XP38={X 318.805969,Y 940.468872,Z 1027.99695,A -176.544083,B 30.8923950,C -165.320572,S 2,T 2,E1 0.0,E2 0.0,E3 0.0,E4 0.0,E5 0.0,E6 0.0}
DECL FDAT FP38={TOOL_NO 9,BASE_NO 3,IPO_FRAME #BASE,POINT2[] " ",TQ_STATE FALSE}
DECL E6POS XPAPOY1={X 116.025192,Y 464.636322,Z 44.8853836,A 90.9894257,B -0.110846877,C -177.937485,S 2,T 34,E1 0.0,E2 0.0,E3 0.0,E4 0.0,E5 0.0,E6 0.0}
DECL FDAT FPAPOY1={TOOL_NO 9,BASE_NO 3,IPO_FRAME #BASE,POINT2[] " ",TQ_STATE FALSE}
DECL E6POS XPAPOY1PRE={X 121.427879,Y 464.439575,Z 194.787933,A 90.9894257,B -0.110846885,C -177.937485,S 2,T 34,E1 0.0,E2 0.0,E3 0.0,E4 0.0,E5 0.0,E6 0.0}
DECL FDAT FPAPOY1PRE={TOOL_NO 9,BASE_NO 3,IPO_FRAME #BASE,POINT2[] " ",TQ_STATE FALSE}
DECL E6POS XPAPOY2PRE={X 230.812134,Y 452.176849,Z 194.359070,A 103.350487,B -0.549977839,C -178.009048,S 2,T 34,E1 0.0,E2 0.0,E3 0.0,E4 0.0,E5 0.0,E6 0.0}
DECL FDAT FPAPOY2PRE={TOOL_NO 9,BASE_NO 3,IPO_FRAME #BASE,POINT2[] " ",TQ_STATE FALSE}
DECL E6POS XPAPOY3PRE={X 511.847778,Y 544.398254,Z 184.744659,A -177.568832,B -1.54007459,C -179.933029,S 2,T 2,E1 0.0,E2 0.0,E3 0.0,E4 0.0,E5 0.0,E6 0.0}
DECL FDAT FPAPOY3PRE={TOOL_NO 9,BASE_NO 3,IPO_FRAME #BASE,POINT2[] " ",TQ_STATE FALSE}
DECL E6POS XPAPOY2={X 225.409439,Y 452.373596,Z 44.4565239,A 103.350487,B -0.549977839,C -178.009048,S 2,T 34,E1 0.0,E2 0.0,E3 0.0,E4 0.0,E5 0.0,E6 0.0}
DECL FDAT FPAPOY2={TOOL_NO 9,BASE_NO 3,IPO_FRAME #BASE,POINT2[] " ",TQ_STATE FALSE}
DECL E6POS XPAPOY4PRE={X 305.220459,Y 691.367798,Z 188.658371,A 179.057358,B -1.53346670,C -179.842529,S 2,T 2,E1 0.0,E2 0.0,E3 0.0,E4 0.0,E5 0.0,E6 0.0}
DECL FDAT FPAPOY4PRE={TOOL_NO 9,BASE_NO 3,IPO_FRAME #BASE,POINT2[] " ",TQ_STATE FALSE}
DECL E6POS XP39={X 320.366150,Y 452.067413,Z 241.559097,A 154.607697,B -1.89703083,C -179.182938,S 2,T 34,E1 0.0,E2 0.0,E3 0.0,E4 0.0,E5 0.0,E6 0.0}
DECL FDAT FP39={TOOL_NO 9,BASE_NO 3,IPO_FRAME #BASE,POINT2[] " ",TQ_STATE FALSE}
DECL E6POS XPAPOY5PRE={X 419.695068,Y 798.575806,Z 173.090652,A -161.858398,B -0.00392377796,C -179.869217,S 2,T 2,E1 0.0,E2 0.0,E3 0.0,E4 0.0,E5 0.0,E6 0.0}
DECL FDAT FPAPOY5PRE={TOOL_NO 9,BASE_NO 3,IPO_FRAME #BASE,POINT2[] " ",TQ_STATE FALSE}
DECL E6POS XPAPOY3={X 507.827423,Y 544.052063,Z 34.7989426,A -177.568832,B -1.54007459,C -179.933029,S 2,T 2,E1 0.0,E2 0.0,E3 0.0,E4 0.0,E5 0.0,E6 0.0}
DECL FDAT FPAPOY3={TOOL_NO 9,BASE_NO 3,IPO_FRAME #BASE,POINT2[] " ",TQ_STATE FALSE}
DECL E6POS XPAPOY6PRE={X 551.381470,Y 880.301,Z 173.191055,A 178.620239,B 0.0400048345,C -179.875427,S 2,T 2,E1 0.0,E2 0.0,E3 0.0,E4 0.0,E5 0.0,E6 0.0}
DECL FDAT FPAPOY6PRE={TOOL_NO 9,BASE_NO 3,IPO_FRAME #BASE,POINT2[] " ",TQ_STATE FALSE}
DECL E6POS XPAPOY7PRE={X 767.409058,Y 914.916077,Z 166.232193,A 126.208084,B 0.123114377,C -179.955719,S 2,T 34,E1 0.0,E2 0.0,E3 0.0,E4 0.0,E5 0.0,E6 0.0}
DECL FDAT FPAPOY7PRE={TOOL_NO 9,BASE_NO 3,IPO_FRAME #BASE,POINT2[] " ",TQ_STATE FALSE}
DECL E6POS XPAPOY4={X 301.200104,Y 691.021606,Z 38.7126617,A 179.057358,B -1.53346670,C -179.842529,S 2,T 2,E1 0.0,E2 0.0,E3 0.0,E4 0.0,E5 0.0,E6 0.0}
DECL FDAT FPAPOY4={TOOL_NO 9,BASE_NO 3,IPO_FRAME #BASE,POINT2[] " ",TQ_STATE FALSE}
DECL E6POS XPAPOY8PRE={X 785.400269,Y 921.451843,Z 168.406891,A 108.921600,B 0.131800815,C -179.993927,S 2,T 34,E1 0.0,E2 0.0,E3 0.0,E4 0.0,E5 0.0,E6 0.0}
DECL FDAT FPAPOY8PRE={TOOL_NO 9,BASE_NO 3,IPO_FRAME #BASE,POINT2[] " ",TQ_STATE FALSE}
DECL E6POS XPAPOY9PRE={X 305.220459,Y 691.367798,Z 188.658371,A 179.057358,B -1.53346670,C -179.842529,S 2,T 2,E1 0.0,E2 0.0,E3 0.0,E4 0.0,E5 0.0,E6 0.0}
DECL FDAT FPAPOY9PRE={TOOL_NO 9,BASE_NO 3,IPO_FRAME #BASE,POINT2[] " ",TQ_STATE FALSE}
DECL E6POS XCAMBIO={X 310.579132,Y 691.828918,Z 388.580,A 178.125076,B -11.0996981,C -166.129044,S 2,T 2,E1 0.0,E2 0.0,E3 0.0,E4 0.0,E5 0.0,E6 0.0}
DECL FDAT FCAMBIO={TOOL_NO 9,BASE_NO 3,IPO_FRAME #BASE,POINT2[] " ",TQ_STATE FALSE}
DECL E6POS XPAPOY10PRE={X 511.847778,Y 544.398254,Z 184.744659,A -177.568832,B -1.54007459,C -179.933029,S 2,T 2,E1 0.0,E2 0.0,E3 0.0,E4 0.0,E5 0.0,E6 0.0}
DECL FDAT FPAPOY10PRE={TOOL_NO 9,BASE_NO 3,IPO_FRAME #BASE,POINT2[] " ",TQ_STATE FALSE}
DECL E6POS XPAPOY5={X 419.791901,Y 798.247253,Z 23.0910492,A -161.858398,B -0.00392381242,C -179.869217,S 2,T 2,E1 0.0,E2 0.0,E3 0.0,E4 0.0,E5 0.0,E6 0.0}
DECL FDAT FPAPOY5={TOOL_NO 9,BASE_NO 3,IPO_FRAME #BASE,POINT2[] " ",TQ_STATE FALSE}
DECL E6POS XPAPOY11PRE={X 511.847778,Y 544.398254,Z 184.744659,A -177.568832,B -1.54007459,C -179.933029,S 2,T 2,E1 0.0,E2 0.0,E3 0.0,E4 0.0,E5 0.0,E6 0.0}
DECL FDAT FPAPOY11PRE={TOOL_NO 9,BASE_NO 3,IPO_FRAME #BASE,POINT2[] " ",TQ_STATE FALSE}
DECL E6POS XPAPOY12PRE={X 305.220459,Y 691.367798,Z 188.658371,A 179.057358,B -1.53346670,C -179.842529,S 2,T 2,E1 0.0,E2 0.0,E3 0.0,E4 0.0,E5 0.0,E6 0.0}
DECL FDAT FPAPOY12PRE={TOOL_NO 9,BASE_NO 3,IPO_FRAME #BASE,POINT2[] " ",TQ_STATE FALSE}
DECL E6POS XPAPOY6={X 551.478333,Y 879.972473,Z 23.1914463,A 178.620239,B 0.0400048159,C -179.875427,S 2,T 2,E1 0.0,E2 0.0,E3 0.0,E4 0.0,E5 0.0,E6 0.0}
DECL FDAT FPAPOY6={TOOL_NO 9,BASE_NO 3,IPO_FRAME #BASE,POINT2[] " ",TQ_STATE FALSE}
DECL E6POS XPAPOY13PRE={X 305.220459,Y 691.367798,Z 188.658371,A 179.057358,B -1.53346670,C -179.842529,S 2,T 2,E1 0.0,E2 0.0,E3 0.0,E4 0.0,E5 0.0,E6 0.0}
DECL FDAT FPAPOY13PRE={TOOL_NO 9,BASE_NO 3,IPO_FRAME #BASE,POINT2[] " ",TQ_STATE FALSE}
DECL E6POS XPAPOY14PRE={X 511.847778,Y 544.398254,Z 184.744659,A -177.568832,B -1.54007459,C -179.933029,S 2,T 2,E1 0.0,E2 0.0,E3 0.0,E4 0.0,E5 0.0,E6 0.0}
DECL FDAT FPAPOY14PRE={TOOL_NO 9,BASE_NO 3,IPO_FRAME #BASE,POINT2[] " ",TQ_STATE FALSE}
DECL E6POS XPAPOY7={X 767.499451,Y 914.609436,Z 26.2325611,A 126.208084,B 0.123114370,C -179.955719,S 2,T 34,E1 0.0,E2 0.0,E3 0.0,E4 0.0,E5 0.0,E6 0.0}
DECL FDAT FPAPOY7={TOOL_NO 9,BASE_NO 3,IPO_FRAME #BASE,POINT2[] " ",TQ_STATE FALSE}
DECL E6POS XPAPOY15PRE={X 511.847778,Y 544.398254,Z 184.744659,A -177.568832,B -1.54007459,C -179.933029,S 2,T 2,E1 0.0,E2 0.0,E3 0.0,E4 0.0,E5 0.0,E6 0.0}
DECL FDAT FPAPOY15PRE={TOOL_NO 9,BASE_NO 3,IPO_FRAME #BASE,POINT2[] " ",TQ_STATE FALSE}
DECL E6POS XPAPOY16PRE={X 305.220459,Y 691.367798,Z 188.658371,A 179.057358,B -1.53346670,C -179.842529,S 2,T 2,E1 0.0,E2 0.0,E3 0.0,E4 0.0,E5 0.0,E6 0.0}
DECL FDAT FPAPOY16PRE={TOOL_NO 9,BASE_NO 3,IPO_FRAME #BASE,POINT2[] " ",TQ_STATE FALSE}
DECL E6POS XPAPOY8={X 785.490662,Y 921.142395,Z 28.4072590,A 108.921600,B 0.131800815,C -179.993927,S 2,T 34,E1 0.0,E2 0.0,E3 0.0,E4 0.0,E5 0.0,E6 0.0}
DECL FDAT FPAPOY8={TOOL_NO 9,BASE_NO 3,IPO_FRAME #BASE,POINT2[] " ",TQ_STATE FALSE}
DECL E6POS XPAPOY17PRE={X 305.220459,Y 691.367798,Z 188.658371,A 179.057358,B -1.53346670,C -179.842529,S 2,T 2,E1 0.0,E2 0.0,E3 0.0,E4 0.0,E5 0.0,E6 0.0}
DECL FDAT FPAPOY17PRE={TOOL_NO 9,BASE_NO 3,IPO_FRAME #BASE,POINT2[] " ",TQ_STATE FALSE}
DECL E6POS XQUITA={X 552.501404,Y 928.451416,Z 732.860352,A 151.668884,B 20.6050854,C 178.563034,S 2,T 34,E1 0.0,E2 0.0,E3 0.0,E4 0.0,E5 0.0,E6 0.0}
DECL FDAT FQUITA={TOOL_NO 9,BASE_NO 3,IPO_FRAME #BASE,POINT2[] " ",TQ_STATE FALSE}
ENDDAT
